{attribute 'qualified_only'}
{attribute 'strict'}
{attribute 'to_string'}
TYPE E_FB_SkillState :
(
    Idle,
    WaitStartAck,
    WaitRunning,
    Running,

    WaitStopAck,
    WaitStopped,

    WaitAbortAck,
    WaitAborted,

    WaitRestartAck,
    WaitRestartStop,
    WaitRestartRunning,

    Done,
    Error
);
END_TYPE

(* stored: Version 1.1.0.1, ProductVersion 3.1.4026.18
   DUT E_FB_SkillState: Id {4e4a8c7a-d4a0-4588-b130-e5e3575789b8} *)
